// TIA Portal V19 export
DATA_BLOCK "Factora Data"   // DB19
{ S7_Optimized_Access := 'TRUE' }
// stored: AutoNumber false, MemoryReserve 0
   VAR RETAIN
      STAT0 : Bool;
      STAT1 : Bool := TRUE;
      STAT2 : Bool := TRUE;
      STAT3 : Bool;
      STAT4 : Bool;
      STAT5 : Bool;
      STAT6 : Bool;
      STAT7 : Bool;
      STAT8 : Bool;
      STAT9 : Bool;
      STAT10 : Bool;
      STAT11 : Bool;
      STAT12 : Bool;
      STAT13 : Bool;
      STAT14 : Bool;
      STAT15 : Bool;
      STAT16 : Word := WORD#16#00A1;
      STAT17 : Word := WORD#16#0006;
      STAT18 : Word;
      STAT19 : Word;
      STAT20 : DWord := DWORD#16#45AE_4A0E;
      STAT21 : DWord;
      STAT22 : DWord;
      STAT23 : DWord;
      STAT24 : Bool;
      STAT25 : Bool := TRUE;
      STAT26 : Bool;
   END_VAR
BEGIN
END_DATA_BLOCK
